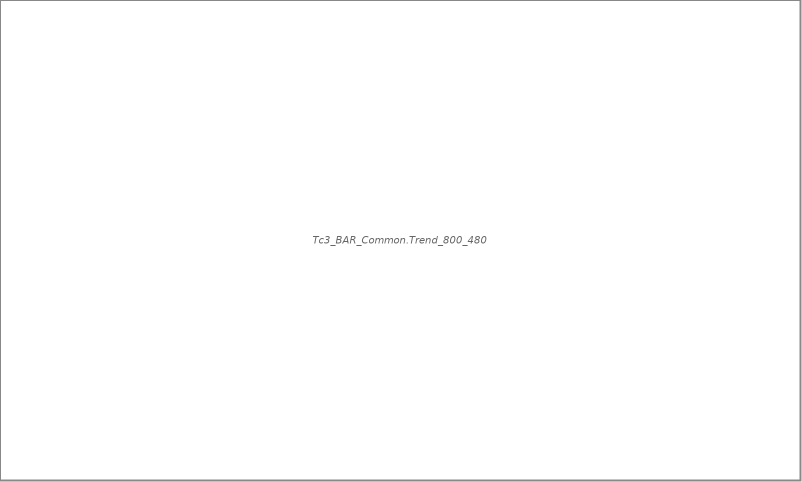
VISUALIZATION TrendsSampleVis  // 802x482
    Frame (0,0 800x480)
        shows Tc3_BAR_Common.Trend_800_480(Header := "Пример названия канала", fb_TrendChanel1 := TrendSample.Var1)
END_VISUALIZATION

(* stored: Version 1.1.0.1, ProductVersion 3.1.4024.2
   Visu TrendsSampleVis: Id {4bf5fb75-393c-44d0-b09c-77c304981b0e} *)
